{attribute 'qualified_only'}
{attribute 'strict'}
TYPE E_Liquids :
(
	water 	:= 0,
	glycol 	:= 1
);
END_TYPE

(* stored: Version 1.1.0.1, ProductVersion 3.1.4024.9
   EnumerationTextList E_Liquids: Id {94f18821-9b9d-4c70-ae71-e6f840948208} *)
